PROGRAM Axis03_Auto
VAR
END_VAR

// NETWORK 1

END_PROGRAM

(* stored: Version 1.1.0.1, ProductVersion 3.1.4024.15
   POU Axis03_Auto: Id {2964529e-7d2c-466b-a161-e686778cebf0}, SpecialFunc None *)
